// Mitsubishi GX Works2 project: PLC_GROUP_04   PLC: FX3G

// global labels: Global1
VAR_GLOBAL
  Work_Day_Light AT Y010 : BOOL;
  Finish_Reset AT M8 : BOOL;
  Check_Ratio AT M1 : BOOL;
  Start_Day AT X010 : BOOL;
  Prep_Start AT X002 : BOOL;
  Prep_Light AT Y005 : BOOL;
  Stock_Flour AT D1100 : REAL;
  Stock_Yeast AT D1110 : REAL;
  Stock_Water AT D1170 : REAL;
  Stock_Oil AT D1130 : REAL;
  Stock_Spice AT D1140 : REAL;
  CS : BOOL;
  Counter_X11 AT CC0 : BOOL;
END_VAR
VAR_GLOBAL CONSTANT
  Constant2 : INT := 2;
  Timer_30 : INT := 30;
END_VAR
VAR_GLOBAL
  Light_Y3 AT Y003 : BOOL;
  Light_Y2 AT Y002 : BOOL;
  CS0 AT CS0 : BOOL;
  Reset_CC0 AT CC0 : BOOL;
  TC2 : BOOL;
  Baking_Timer AT TC2 : BOOL;
  Baking_Light AT Y004 : BOOL;
END_VAR
VAR_GLOBAL CONSTANT
  Timer_40 : INT := 40;
END_VAR
VAR_GLOBAL
  Done_Swelling AT Y003 : BOOL;
  Done_Swelling2 AT Y002 : BOOL;
  Quality_Check AT X003 : BOOL;
  Save_Analog_Value AT D3000 : REAL;
  analogInput AT D8000 : REAL;
END_VAR
VAR_GLOBAL CONSTANT
  GreaterThen1 : INT := 400;
END_VAR
VAR_GLOBAL
  analogInput2 AT D8005 : REAL;
END_VAR
VAR_GLOBAL CONSTANT
  LowerThen5 : INT := 2000;
END_VAR
VAR_GLOBAL
  Timer_Qulity_Light AT TC8 : BOOL;
END_VAR
VAR_GLOBAL CONSTANT
  Timer_50 : INT := 50;
END_VAR
VAR_GLOBAL
  Quality_Light AT Y006 : BOOL;
  Prep_Light_Timer AT TC0 : BOOL;
END_VAR
VAR_GLOBAL CONSTANT
  Timer30 : INT := 30;
END_VAR
VAR_GLOBAL
  Prep_Input AT Y005 : BOOL;
  Take_Flour AT D1100 : REAL;
END_VAR
VAR_GLOBAL CONSTANT
  KgFlour : REAL := 100;
END_VAR
VAR_GLOBAL
  New_Flour_Amount AT D1100 : REAL;
  Take_Oil AT D1130 : REAL;
END_VAR
VAR_GLOBAL CONSTANT
  LiterOil : REAL := 30;
END_VAR
VAR_GLOBAL
  New_Oil_Amount AT D1130 : REAL;
  Take_Spice AT D1140 : REAL;
END_VAR
VAR_GLOBAL CONSTANT
  KgSpice : REAL := 10;
END_VAR
VAR_GLOBAL
  New_Spice_Amount AT D1140 : REAL;
  Take_Water AT D1120 : REAL;
END_VAR
VAR_GLOBAL CONSTANT
  LiterWater : REAL := 50;
END_VAR
VAR_GLOBAL
  New_Water_Amount AT D1120 : REAL;
  Take_Yeast AT D1110 : REAL;
END_VAR
VAR_GLOBAL CONSTANT
  KgYeast : REAL := 20;
END_VAR
VAR_GLOBAL
  New_Yeast_Amount AT D1110 : REAL;
  Start_Kneading AT X001 : BOOL;
  End_Kneading AT X011 : BOOL;
  Kneading_Light AT Y001 : BOOL;
  Flour_Stock AT D1100 : REAL;
END_VAR
VAR_GLOBAL CONSTANT
  Flour_Limit : REAL := 100;
END_VAR
VAR_GLOBAL
  Oil_Ratio AT D1100 : REAL;
END_VAR
VAR_GLOBAL CONSTANT
  Flour_Oil_R : REAL := 0.3;
END_VAR
VAR_GLOBAL
  Oil_Expected AT D1200 : REAL;
  Oil_Check AT D1200 : REAL;
  Spice_ratio AT D1100 : REAL;
END_VAR
VAR_GLOBAL CONSTANT
  Flour_Spice_R : REAL := 0.1;
END_VAR
VAR_GLOBAL
  Spice_Expected AT D1240 : REAL;
  Oil_light AT M13 : BOOL;
  Spice_Check AT D1240 : REAL;
  Spice_Light AT M14 : BOOL;
  Water_Ratio AT D1100 : REAL;
END_VAR
VAR_GLOBAL CONSTANT
  Flour_Water_R : REAL := 0.5;
END_VAR
VAR_GLOBAL
  Water_Expected AT D1220 : REAL;
  Water_Check AT D1220 : REAL;
  Water_Light AT M15 : BOOL;
  Yeast_Ratio AT D1100 : REAL;
END_VAR
VAR_GLOBAL CONSTANT
  Flour_Yeast_R : REAL := 0.2;
END_VAR
VAR_GLOBAL
  Yeast_Expected AT D1210 : REAL;
  Yeast_Check AT D1210 : REAL;
  Yeast_Light AT M16 : BOOL;
  Oil_OK AT M13 : BOOL;
  Spice_OK AT M14 : BOOL;
  Water_OK AT M15 : BOOL;
  Yeast_OK AT M16 : BOOL;
  Emergency_Switch AT X007 : BOOL;
  Day_Light AT Y010 : BOOL;
  Keep_Light AT Y010 : BOOL;
  ananlog_Output AT M11 : BOOL;
  Output_LT AT M11 : BOOL;
  analog_Output AT M10 : BOOL;
  Output_HT AT M10 : BOOL;
  ananlog_Output2 AT M11 : BOOL;
  analog_Output2 AT M11 : BOOL;
  Resault AT M13 : BOOL;
  Flour1 AT M12 : BOOL;
  Oil1 AT M14 : BOOL;
  Spice1 AT M15 : BOOL;
  Water1 AT M16 : BOOL;
  Yeast1 AT M17 : BOOL;
  fixOutput2 AT M19 : BOOL;
  fixOutput1 AT M18 : BOOL;
  Oil_input AT D1145 : REAL;
  water_input AT D1147 : REAL;
  Flour_input AT D1156 : REAL;
  spice_input AT D1166 : REAL;
  yeast_input AT D1677 : REAL;
  alll_OK AT M13 : BOOL;
  Light_timer AT TC4 : BOOL;
  Prep_Light_Timer_TS AT TS0 : BOOL;
  Stop_Count AT CS0 : BOOL;
  Stop_Baking AT TS2 : BOOL;
  Stop_Kneading AT M20 : BOOL;
  Flash_Y2 AT TC4 : BOOL;
END_VAR
VAR_GLOBAL CONSTANT
  Flash_Time : INT := 10;
END_VAR
VAR_GLOBAL
  flashy2 AT TS4 : BOOL;
  F2 AT M8 : BOOL;
  Flash_Y3 AT TC5 : BOOL;
END_VAR
VAR_GLOBAL CONSTANT
  Flash_Time2 : INT := 10;
END_VAR
VAR_GLOBAL
  flashy3 AT TS5 : BOOL;
  start_count AT CS0 : BOOL;
  Count_1 AT M140 : BOOL;
  Count_2 AT M150 : BOOL;
END_VAR
VAR_GLOBAL CONSTANT
  Timer3 : INT := 30;
END_VAR
VAR_GLOBAL
  timeY2 AT TC7 : BOOL;
  End_Day AT M0 : BOOL;
  End_Day_Light AT M25 : BOOL;
  Stock_Done AT M23 : BOOL;
  NoFlour AT M100 : BOOL;
  End_Light_10 AT CS2 : BOOL;
  Light AT M30 : BOOL;
  Light10Y AT TS2 : BOOL;
  Light1 AT TC2 : BOOL;
END_VAR
VAR_GLOBAL CONSTANT
  LightNum : INT := 5;
END_VAR
VAR_GLOBAL
  Light2 AT TC3 : BOOL;
  Light01 AT M31 : BOOL;
  Light10Ytwo AT TS2 : BOOL;
  End_Light10 AT CC2 : BOOL;
END_VAR
VAR_GLOBAL CONSTANT
  NumY10 : INT := 6;
END_VAR
VAR_GLOBAL
  Kneading AT M80 : BOOL;
  Press_1 AT M60 : BOOL;
  Press_2 AT M55 : BOOL;
  Test_Ratio AT M77 : BOOL;
  Baking AT M76 : BOOL;
  Finish_Kneading AT TS7 : BOOL;
  Baking_Time AT TC10 : BOOL;
  Quality_Off AT TS8 : BOOL;
  Analog_Input AT D8281 : INT;
END_VAR
VAR_GLOBAL CONSTANT
  add_210 : REAL := 210;
END_VAR
VAR_GLOBAL
  Shelf AT D7998 : REAL;
  Light10Y2 AT TS3 : BOOL;
END_VAR
VAR_GLOBAL CONSTANT
  Count10 : INT := 6;
END_VAR
VAR_GLOBAL
  Finish_Baking AT TS10 : BOOL;
  Flour_Tank AT D7666 : REAL;
  Oil_Tank AT D7555 : REAL;
  Spice_Tank AT D7444 : REAL;
  Water_Tank AT D7333 : REAL;
  Yeast_Tank AT D7222 : REAL;
END_VAR
VAR_GLOBAL CONSTANT
  Constant_100 : REAL := 100;
  Contant_30 : REAL := 30;
  Constant_50 : REAL := 50;
  Constant_20 : REAL := 20;
  Constant_210 : REAL := 210;
END_VAR
VAR_GLOBAL
  Kneading_Phase AT D7111 : REAL;
  Storage AT D1212 : REAL;
  Baking_Phase AT M76 : BOOL;
  Baking_Pan AT D7212 : REAL;
END_VAR

// task Task_01 (event TRUE, interval 0, priority 31): POU_01

PROGRAM POU_01
(* structured ladder/FBD written out as ST: instructions are called as NAME(EN, inputs, outputs); _pN, _eN, _tN stand for wires *)
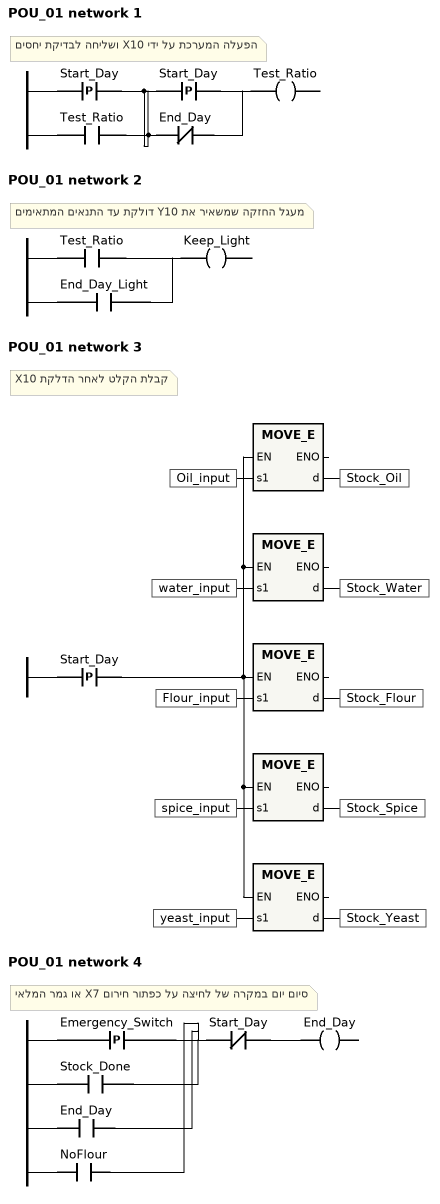
(* network 1 *)
(* הפעלה המערכת על ידי X10 ושליחה לבדיקת יחסים *)
_p1 := LDP(TRUE, Start_Day) OR Test_Ratio;
Test_Ratio := (_p1 AND LDP(TRUE, Start_Day)) OR (_p1 AND NOT End_Day);
(* network 2 *)
(* מעגל החזקה שמשאיר את Y10 דולקת עד התנאים המתאימים *)
Keep_Light := Test_Ratio OR End_Day_Light;
(* network 3 *)
(* קבלת הקלט לאחר הדלקת X10 *)
_p1 := LDP(TRUE, Start_Day);
MOVE_E(_p1, Oil_input, Stock_Oil);
MOVE_E(_p1, water_input, Stock_Water);
MOVE_E(_p1, Flour_input, Stock_Flour);
MOVE_E(_p1, spice_input, Stock_Spice);
MOVE_E(_p1, yeast_input, Stock_Yeast);
(* network 4 *)
(* סיום יום במקרה של לחיצה על כפתור חירום X7 או גמר המלאי *)
End_Day := (LDP(TRUE, Emergency_Switch) OR Stock_Done OR End_Day OR NoFlour) AND NOT Start_Day;
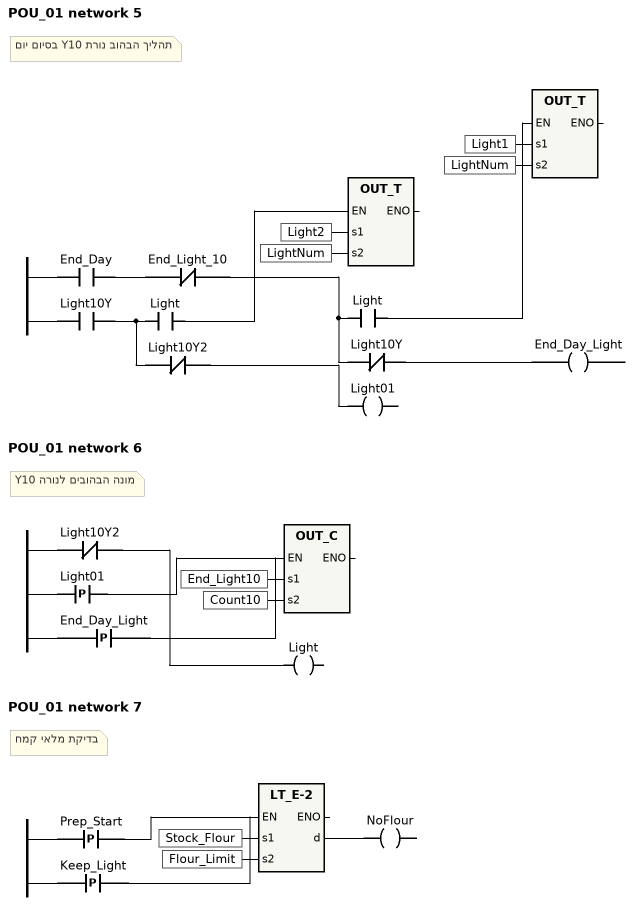
(* network 5 *)
(* תהליך הבהוב נורת Y10 בסיום יום *)
_p1 := End_Day AND NOT End_Light_10;
OUT_T(_p1 AND Light, Light1, LightNum);
End_Day_Light := _p1 AND NOT Light10Y;
OUT_T(Light10Y AND Light, Light2, LightNum);
Light01 := Light10Y AND NOT Light10Y2;
(* network 6 *)
(* מונה הבהובים לנורה Y10 *)
Light := NOT Light10Y2;
OUT_C(LDP(TRUE, Light01) OR LDP(TRUE, End_Day_Light), End_Light10, Count10);
(* network 7 *)
(* בדיקת מלאי קמח *)
LT_E(LDP(TRUE, Prep_Start) OR LDP(TRUE, Keep_Light), Stock_Flour, Flour_Limit, _t1);
NoFlour := _t1;
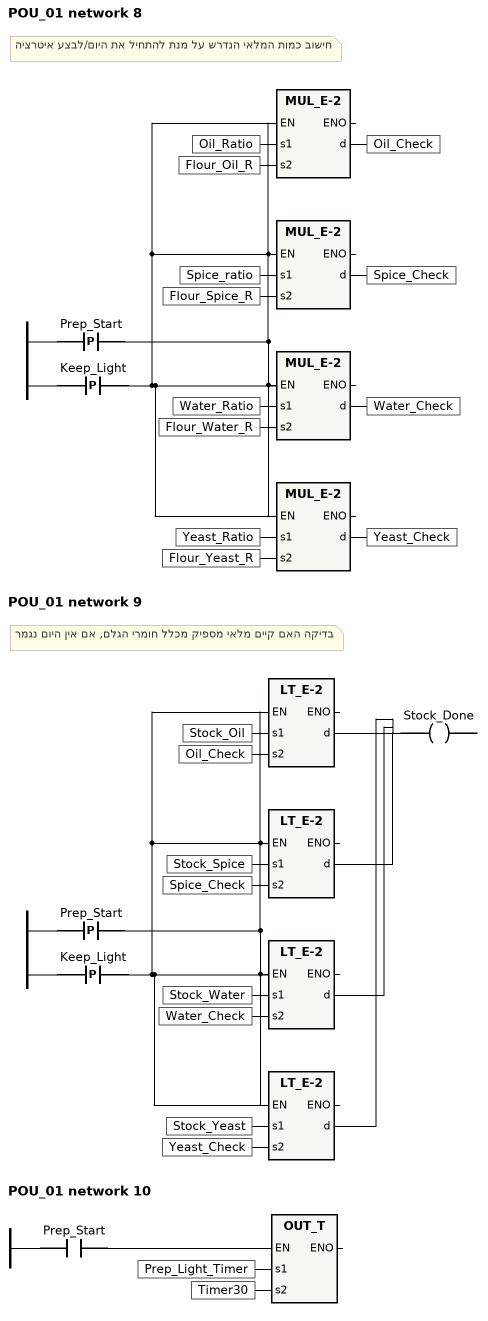
(* network 8 *)
(* חישוב כמות המלאי הנדרש על מנת להתחיל את היום/לבצע איטרציה *)
_p1 := LDP(TRUE, Prep_Start) OR LDP(TRUE, Keep_Light);
MUL_E(_p1, Oil_Ratio, Flour_Oil_R, Oil_Check);
MUL_E(_p1, Spice_ratio, Flour_Spice_R, Spice_Check);
MUL_E(_p1, Water_Ratio, Flour_Water_R, Water_Check);
MUL_E(_p1, Yeast_Ratio, Flour_Yeast_R, Yeast_Check);
(* network 9 *)
(* בדיקה האם קיים מלאי מספיק מכלל חומרי הגלם, אם אין היום נגמר *)
_p1 := LDP(TRUE, Prep_Start) OR LDP(TRUE, Keep_Light);
LT_E(_p1, Stock_Oil, Oil_Check, _t2);
LT_E(_p1, Stock_Spice, Spice_Check, _t3);
LT_E(_p1, Stock_Water, Water_Check, _t4);
LT_E(_p1, Stock_Yeast, Yeast_Check, _t5);
Stock_Done := _t2 OR _t3 OR _t4 OR _t5;
(* network 10 *)
OUT_T(Prep_Start, Prep_Light_Timer, Timer30);
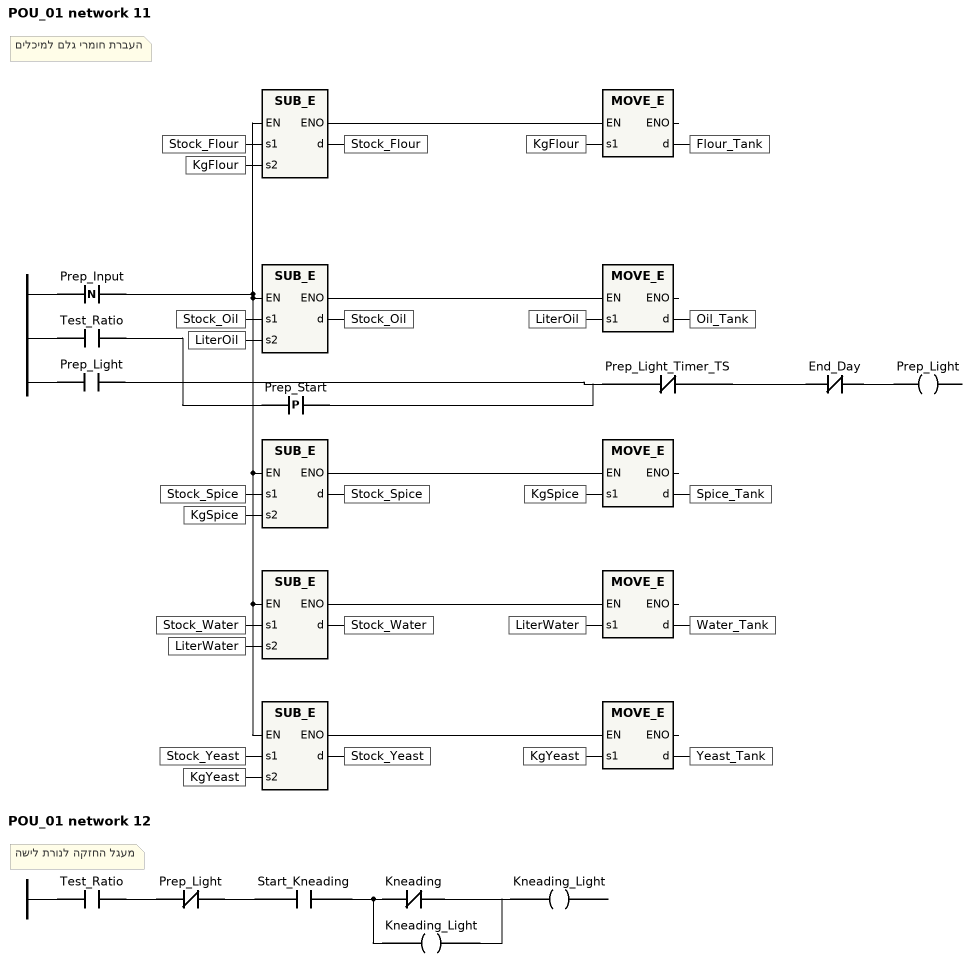
(* network 11 *)
(* העברת חומרי גלם למיכלים *)
_p1 := LDF(TRUE, Prep_Input);
_e2 := SUB_E(_p1, Stock_Flour, KgFlour, Stock_Flour);
MOVE_E(_e2, KgFlour, Flour_Tank);
_e3 := SUB_E(_p1, Stock_Oil, LiterOil, Stock_Oil);
MOVE_E(_e3, LiterOil, Oil_Tank);
_e4 := SUB_E(_p1, Stock_Spice, KgSpice, Stock_Spice);
MOVE_E(_e4, KgSpice, Spice_Tank);
_e5 := SUB_E(_p1, Stock_Water, LiterWater, Stock_Water);
MOVE_E(_e5, LiterWater, Water_Tank);
_e6 := SUB_E(_p1, Stock_Yeast, KgYeast, Stock_Yeast);
MOVE_E(_e6, KgYeast, Yeast_Tank);
Prep_Light := (((Test_Ratio AND LDP(TRUE, Prep_Start)) OR Prep_Light) AND NOT Prep_Light_Timer_TS) AND NOT End_Day;
(* network 12 *)
(* מעגל החזקה לנורת לישה *)
_p1 := Test_Ratio AND NOT Prep_Light AND Start_Kneading;
Kneading_Light := _p1;
Kneading_Light := (_p1 AND NOT Kneading) OR _p1;
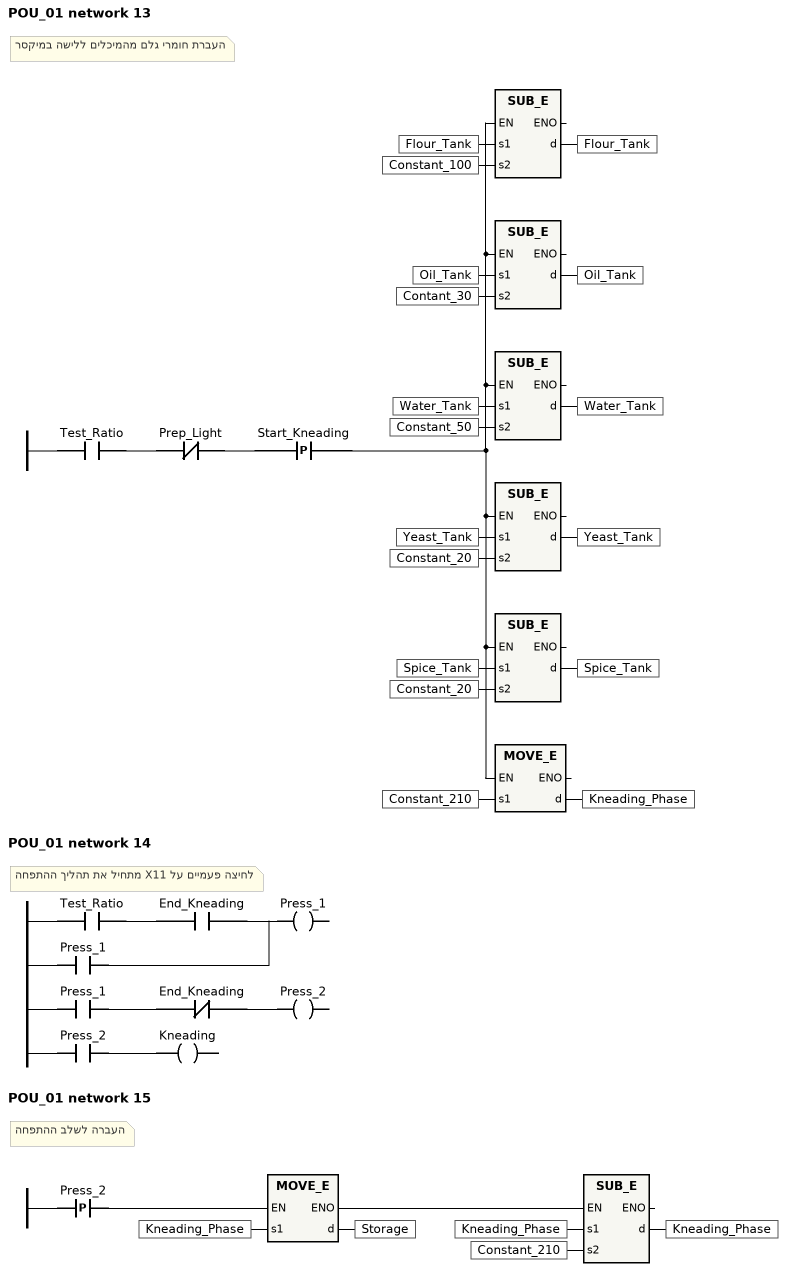
(* network 13 *)
(* העברת חומרי גלם מהמיכלים ללישה במיקסר *)
_p1 := Test_Ratio AND NOT Prep_Light AND LDP(TRUE, Start_Kneading);
SUB_E(_p1, Flour_Tank, Constant_100, Flour_Tank);
SUB_E(_p1, Oil_Tank, Contant_30, Oil_Tank);
SUB_E(_p1, Water_Tank, Constant_50, Water_Tank);
SUB_E(_p1, Yeast_Tank, Constant_20, Yeast_Tank);
SUB_E(_p1, Spice_Tank, Constant_20, Spice_Tank);
MOVE_E(_p1, Constant_210, Kneading_Phase);
(* network 14 *)
(* לחיצה פעמיים על X11 מתחיל את תהליך ההתפחה *)
Press_1 := (Test_Ratio AND End_Kneading) OR Press_1;
Press_2 := Press_1 AND NOT End_Kneading;
Kneading := Press_2;
(* network 15 *)
(* העברה לשלב ההתפחה *)
_e1 := MOVE_E(LDP(TRUE, Press_2), Kneading_Phase, Storage);
SUB_E(_e1, Kneading_Phase, Constant_210, Kneading_Phase);
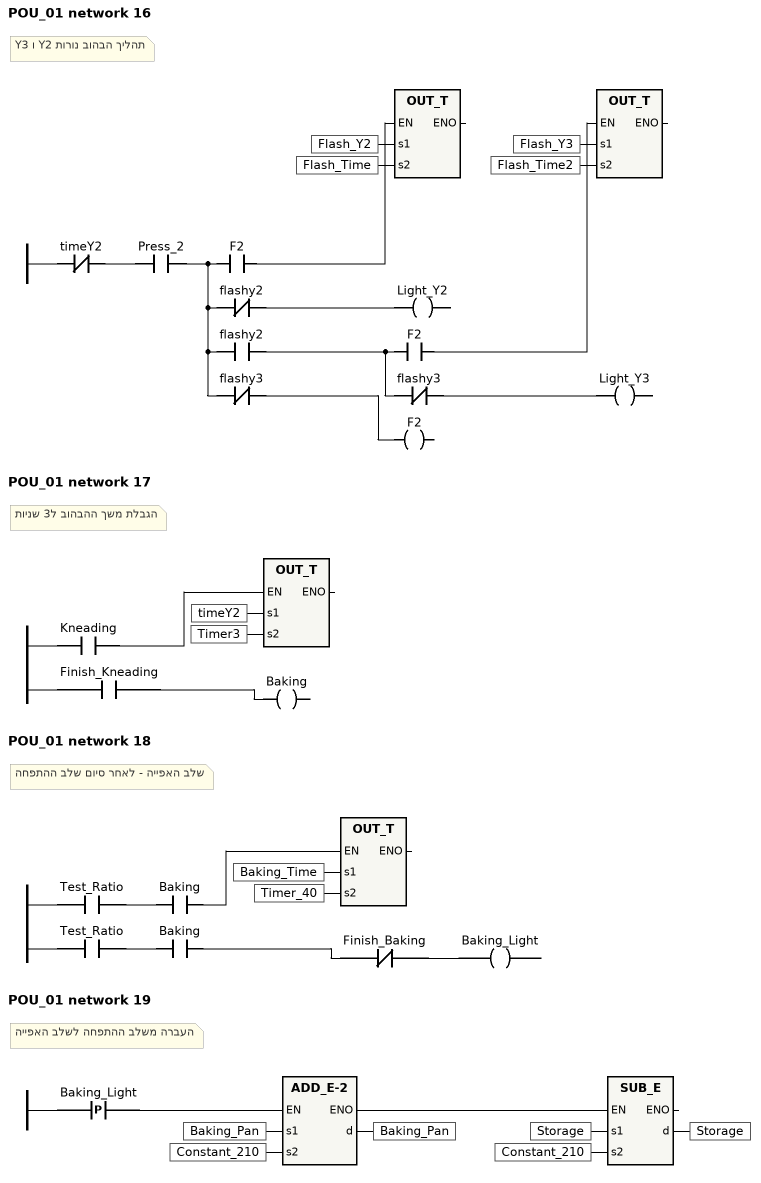
(* network 16 *)
(* תהליך הבהוב נורות Y2 ו Y3 *)
_p1 := NOT timeY2 AND Press_2;
OUT_T(_p1 AND F2, Flash_Y2, Flash_Time);
Light_Y2 := _p1 AND NOT flashy2;
_p2 := _p1 AND flashy2;
OUT_T(_p2 AND F2, Flash_Y3, Flash_Time2);
Light_Y3 := _p2 AND NOT flashy3;
F2 := _p1 AND NOT flashy3;
(* network 17 *)
(* הגבלת משך ההבהוב ל3 שניות *)
OUT_T(Kneading, timeY2, Timer3);
Baking := Finish_Kneading;
(* network 18 *)
(* שלב האפייה - לאחר סיום שלב ההתפחה *)
OUT_T(Test_Ratio AND Baking, Baking_Time, Timer_40);
Baking_Light := Test_Ratio AND Baking AND NOT Finish_Baking;
(* network 19 *)
(* העברה משלב ההתפחה לשלב האפייה *)
_e1 := ADD_E(LDP(TRUE, Baking_Light), Baking_Pan, Constant_210, Baking_Pan);
SUB_E(_e1, Storage, Constant_210, Storage);
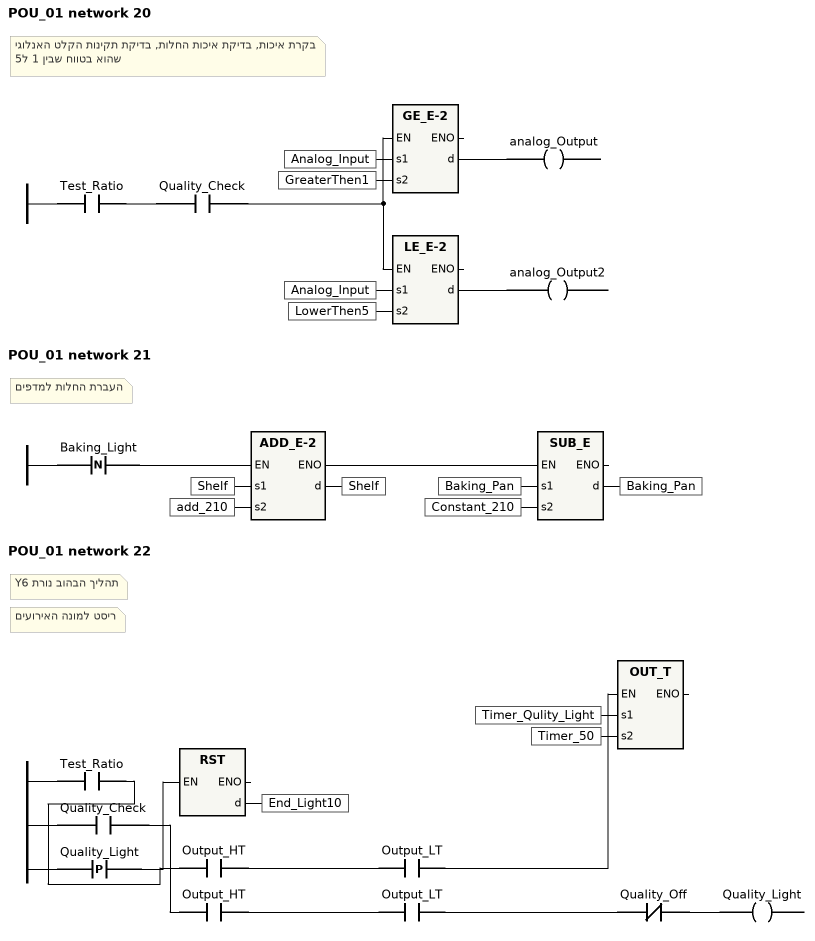
(* network 20 *)
(* בקרת איכות, בדיקת איכות החלות, בדיקת תקינות הקלט האנלוגי שהוא בטווח שבין 1 ל5 *)
_p1 := Test_Ratio AND Quality_Check;
GE_E(_p1, Analog_Input, GreaterThen1, _t2);
analog_Output := _t2;
LE_E(_p1, Analog_Input, LowerThen5, _t3);
analog_Output2 := _t3;
(* network 21 *)
(* העברת החלות למדפים *)
_e1 := ADD_E(LDF(TRUE, Baking_Light), Shelf, add_210, Shelf);
SUB_E(_e1, Baking_Pan, Constant_210, Baking_Pan);
(* network 22 *)
(* תהליך הבהוב נורת Y6 *)
(* ריסט למונה האירועים *)
OUT_T(Test_Ratio AND Output_HT AND Output_LT, Timer_Qulity_Light, Timer_50);
Quality_Light := Quality_Check AND Output_HT AND Output_LT AND NOT Quality_Off;
RST(LDP(TRUE, Quality_Light), End_Light10);
END_PROGRAM
